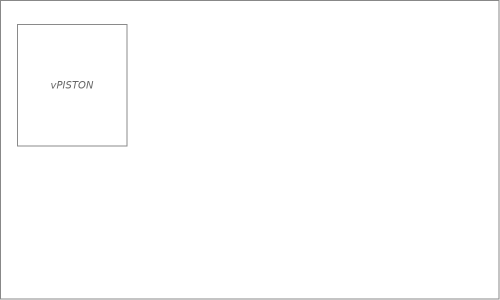
VISUALIZATION vSTATIONS  // 500x300
    Frame (17,24 110x122)
        shows vPISTON(PIST1 := PIST1)
END_VISUALIZATION

(* stored: Version 1.1.0.1, ProductVersion 3.1.4024.12
   Visu vSTATIONS: Id {9b3a510f-13aa-4e9a-bbe4-7a1c9102ea84} *)
